# EPICS autosave request: tests/testfiles/cfg/SF_Acc_PV.req
$(SYS)-RMSM:SM-SET
$(SYS)-RSYS:REQUIRED-OP
$(SYS)-RSYS:SET-BEAM-PHASE
$(SYS)-RSYS:SET-ACC-VOLT
